// TIA Portal V19 export
VAR_GLOBAL   // PLC tag table "conveyor-0"
   "Start Button 0" AT %I0.0 : Bool;
   "Belt Conveyor (4m) 0" AT %Q0.0 : Bool;
   "memedge0-0" AT %M0.0 : Bool;
   "memedge0-1" AT %M0.1 : Bool;
   "memedge0-2" AT %M0.2 : Bool;
   "mem0-start" AT %M0.3 : Bool;
   "memory0-0" AT %M0.4 : Bool;
END_VAR
